FUNCTION SPLIT_DWORD_INTO_QUARTERS (* this Function extracts the 16 QUARTER BYTE from a dword *)
  (* Standard: 61499-1; Description: Copyright (c) 2024 HR Agrartechnik GmbH This program and the accompanying materials are made available under the terms of the Eclipse Public License 2.0 which is available at https://www.eclipse.org/legal/epl-2.0/ SPDX-License-Identifier: EPL-2.0 *)
  (* Version 3.0.1, 2026-09-29, Martin Jobst, fix ST package declaration *)
  (* Version 3.0, 2025-04-14, Patrick Aigner, changed package *)
  (* Version 1.1, 2024-07-24, Moritz Ortmeier, HR Agrartechnik, rename Function and change Output Variables *)
  (* Version 1.0, 2024-02-22, Franz Höpfinger, HR Agrartechnik, initial Implementation *)
  PACKAGE eclipse4diac::utils::splitting;
  IMPORT eclipse4diac::utils::const::quarterconst;
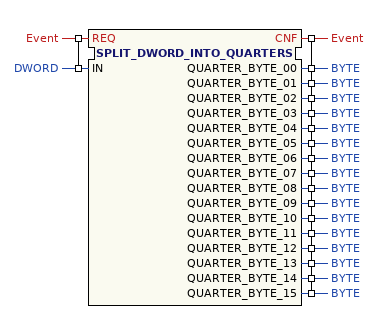
  EVENT_INPUT
    REQ WITH IN;
  END_EVENT
  EVENT_OUTPUT
    CNF WITH QUARTER_BYTE_00, QUARTER_BYTE_01, QUARTER_BYTE_02, QUARTER_BYTE_03, QUARTER_BYTE_04, QUARTER_BYTE_05, QUARTER_BYTE_06, QUARTER_BYTE_07, QUARTER_BYTE_08, QUARTER_BYTE_09, QUARTER_BYTE_10, QUARTER_BYTE_11, QUARTER_BYTE_12, QUARTER_BYTE_13, QUARTER_BYTE_14, QUARTER_BYTE_15;
  END_EVENT
  VAR_INPUT
    IN : DWORD;
  END_VAR
  VAR_OUTPUT
    QUARTER_BYTE_00 : BYTE;
    QUARTER_BYTE_01 : BYTE;
    QUARTER_BYTE_02 : BYTE;
    QUARTER_BYTE_03 : BYTE;
    QUARTER_BYTE_04 : BYTE;
    QUARTER_BYTE_05 : BYTE;
    QUARTER_BYTE_06 : BYTE;
    QUARTER_BYTE_07 : BYTE;
    QUARTER_BYTE_08 : BYTE;
    QUARTER_BYTE_09 : BYTE;
    QUARTER_BYTE_10 : BYTE;
    QUARTER_BYTE_11 : BYTE;
    QUARTER_BYTE_12 : BYTE;
    QUARTER_BYTE_13 : BYTE;
    QUARTER_BYTE_14 : BYTE;
    QUARTER_BYTE_15 : BYTE;
  END_VAR
  BODY IN ST:
PACKAGE eclipse4diac::utils::splitting;

IMPORT eclipse4diac::utils::const::quarterconst;

(* this Function extracts the 16 QUARTER BYTE from a dword *)
FUNCTION SPLIT_DWORD_INTO_QUARTERS

VAR_INPUT
	IN : DWORD;
END_VAR

VAR_OUTPUT
	QUARTER_BYTE_00 : BYTE;
	QUARTER_BYTE_01 : BYTE;
	QUARTER_BYTE_02 : BYTE;
	QUARTER_BYTE_03 : BYTE;
	QUARTER_BYTE_04 : BYTE;
	QUARTER_BYTE_05 : BYTE;
	QUARTER_BYTE_06 : BYTE;
	QUARTER_BYTE_07 : BYTE;
	QUARTER_BYTE_08 : BYTE;
	QUARTER_BYTE_09 : BYTE;
	QUARTER_BYTE_10 : BYTE;
	QUARTER_BYTE_11 : BYTE;
	QUARTER_BYTE_12 : BYTE;
	QUARTER_BYTE_13 : BYTE;
	QUARTER_BYTE_14 : BYTE;
	QUARTER_BYTE_15 : BYTE;
END_VAR

QUARTER_BYTE_00 := DWORD_TO_BYTE(SHR(IN AND quarterconst::DWORD_QUARTER_00, quarterconst::SHIFT_QUARTER_00));
QUARTER_BYTE_01 := DWORD_TO_BYTE(SHR(IN AND quarterconst::DWORD_QUARTER_01, quarterconst::SHIFT_QUARTER_01));
QUARTER_BYTE_02 := DWORD_TO_BYTE(SHR(IN AND quarterconst::DWORD_QUARTER_02, quarterconst::SHIFT_QUARTER_02));
QUARTER_BYTE_03 := DWORD_TO_BYTE(SHR(IN AND quarterconst::DWORD_QUARTER_03, quarterconst::SHIFT_QUARTER_03));
QUARTER_BYTE_04 := DWORD_TO_BYTE(SHR(IN AND quarterconst::DWORD_QUARTER_04, quarterconst::SHIFT_QUARTER_04));
QUARTER_BYTE_05 := DWORD_TO_BYTE(SHR(IN AND quarterconst::DWORD_QUARTER_05, quarterconst::SHIFT_QUARTER_05));
QUARTER_BYTE_06 := DWORD_TO_BYTE(SHR(IN AND quarterconst::DWORD_QUARTER_06, quarterconst::SHIFT_QUARTER_06));
QUARTER_BYTE_07 := DWORD_TO_BYTE(SHR(IN AND quarterconst::DWORD_QUARTER_07, quarterconst::SHIFT_QUARTER_07));
QUARTER_BYTE_08 := DWORD_TO_BYTE(SHR(IN AND quarterconst::DWORD_QUARTER_08, quarterconst::SHIFT_QUARTER_08));
QUARTER_BYTE_09 := DWORD_TO_BYTE(SHR(IN AND quarterconst::DWORD_QUARTER_09, quarterconst::SHIFT_QUARTER_09));
QUARTER_BYTE_10 := DWORD_TO_BYTE(SHR(IN AND quarterconst::DWORD_QUARTER_10, quarterconst::SHIFT_QUARTER_10));
QUARTER_BYTE_11 := DWORD_TO_BYTE(SHR(IN AND quarterconst::DWORD_QUARTER_11, quarterconst::SHIFT_QUARTER_11));
QUARTER_BYTE_12 := DWORD_TO_BYTE(SHR(IN AND quarterconst::DWORD_QUARTER_12, quarterconst::SHIFT_QUARTER_12));
QUARTER_BYTE_13 := DWORD_TO_BYTE(SHR(IN AND quarterconst::DWORD_QUARTER_13, quarterconst::SHIFT_QUARTER_13));
QUARTER_BYTE_14 := DWORD_TO_BYTE(SHR(IN AND quarterconst::DWORD_QUARTER_14, quarterconst::SHIFT_QUARTER_14));
QUARTER_BYTE_15 := DWORD_TO_BYTE(SHR(IN AND quarterconst::DWORD_QUARTER_15, quarterconst::SHIFT_QUARTER_15));
END_FUNCTION
  END_BODY
END_FUNCTION
